PROGRAM PeriodicMesure
VAR
	fbSQLDatabase : FB_SQLDatabaseEvt(sNetID := '', tTimeout := T#5S);

	fbSQLCommand : FB_SQLCommandEvt(sNetID := '', tTimeOut := T#5S);

	step : (OPEN_CONNECTION, CREATE_MESURE, INSERT_MESURE, CLOSE_CONNECTION, FINISH) := OPEN_CONNECTION;
	CMD25 : STRING(255);
	CMD20 : STRING(255);
	CMD : STRING(1000);
	
	rVR25True : REAL;
	rVR20True : REAL;
	
	jsonString : STRING(5000);
	
	
END_VAR

CASE step OF
	
	OPEN_CONNECTION:

		IF fbSQLDatabase.Connect(1) THEN
			step := CREATE_MESURE;
		END_IF
		
	CREATE_MESURE:
		IF fbSQLDatabase.CreateCmd(ADR(fbSQLCommand)) THEN
			step := INSERT_MESURE;
		END_IF
		
	INSERT_MESURE:
		
		// Convert raw value to mm/s
	
		rVR25True := GVL.iVR25Value * 0.000488296151 * 1.5625;
		rVR20True := GVL.iVR20Value * 0.000488296151 * 1.25;
		
		// Creating jsonString VR25
		
		jsonString := CONCAT('$'{"type":"', GVL.sTypeVR25);
		jsonString := CONCAT(jsonString, '","uom":"');
		jsonString := CONCAT(jsonString, GVL.sUomVR25);
		jsonString := CONCAT(jsonString, '","value":');
		jsonString := CONCAT(jsonString, REAL_TO_STRING(rVR25True));
		jsonString := CONCAT(jsonString, '}$'');
		
		// Creating SQL Query VR25
	
		CMD25 := CONCAT('INSERT INTO Tag (timestampStart, json_data, id_client, id_machine, id_daq, id_plant, id_image) VALUES (',ULINT_TO_STRING(F_GetSystemTime()));
		CMD25 := CONCAT(CMD25, ',');
		CMD25 := CONCAT(CMD25, jsonString);
		CMD25 := CONCAT(CMD25, ',');
		CMD25 := CONCAT(CMD25, INT_TO_STRING(GVL.iIDClient));
		CMD25 := CONCAT(CMD25, ',');
		CMD25 := CONCAT(CMD25, INT_TO_STRING(GVL.iIDMachine));
		CMD25 := CONCAT(CMD25, ',');
		CMD25 := CONCAT(CMD25, INT_TO_STRING(GVL.iIDDAQVR25));
		CMD25 := CONCAT(CMD25, ',');
		CMD25 := CONCAT(CMD25, INT_TO_STRING(GVL.iIDPlant));
		CMD25 := CONCAT(CMD25, ',');
		CMD25 := CONCAT(CMD25, INT_TO_STRING(GVL.iIDImageVR25));
		CMD25 := CONCAT(CMD25, ');');
		
		// Creating jsonString VR20
		
		jsonString := CONCAT('$'{"type":"', GVL.sTypeVR20);
		jsonString := CONCAT(jsonString, '","uom":"');
		jsonString := CONCAT(jsonString, GVL.sUomVR20);
		jsonString := CONCAT(jsonString, '","value":');
		jsonString := CONCAT(jsonString, REAL_TO_STRING(rVR20True));
		jsonString := CONCAT(jsonString, '}$'');
		
		// Creating SQL Query VR20
		
		CMD20 := CONCAT('INSERT INTO Tag (timestampStart, json_data, id_client, id_machine, id_daq, id_plant, id_image) VALUES (',ULINT_TO_STRING(F_GetSystemTime()));
		CMD20 := CONCAT(CMD20, ',');
		CMD20 := CONCAT(CMD20, jsonString);
		CMD20 := CONCAT(CMD20, ',');
		CMD20 := CONCAT(CMD20, INT_TO_STRING(GVL.iIDClient));
		CMD20 := CONCAT(CMD20, ',');
		CMD20 := CONCAT(CMD20, INT_TO_STRING(GVL.iIDMachine));
		CMD20 := CONCAT(CMD20, ',');
		CMD20 := CONCAT(CMD20, INT_TO_STRING(GVL.iIDDAQVR20));
		CMD20 := CONCAT(CMD20, ',');
		CMD20 := CONCAT(CMD20, INT_TO_STRING(GVL.iIDPlant));
		CMD20 := CONCAT(CMD20, ',');
		CMD20 := CONCAT(CMD20, INT_TO_STRING(GVL.iIDImageVR20));
		CMD20 := CONCAT(CMD20, ');');
		
		CONCAT2(ADR(CMD25), ADR(CMD20), ADR(CMD), SIZEOF(CMD));
		
		IF fbSQLCommand.Execute(ADR(CMD), SIZEOF(CMD)) THEN
			step := CLOSE_CONNECTION;
		END_IF
	
	CLOSE_CONNECTION:
		IF fbSQLDatabase.Disconnect() THEN
			step := FINISH;
		END_IF
		
	FINISH:
		step := OPEN_CONNECTION; 

		
END_CASE

METHOD isfinished : BOOL
IF step = FINISH THEN
	isfinished := TRUE;
ELSE
	isfinished := FALSE;
END_IF
END_METHOD

END_PROGRAM

(* stored: Version 1.1.0.1, ProductVersion 3.1.4024.12
   POU PeriodicMesure: Id {bd7a1e3e-4ebf-41f5-baf8-0d762dd80132}, SpecialFunc None
   Method isfinished: Id {15a57adf-def9-416d-bd35-5116e158f3a0} *)
